// TIA Portal V19 export
DATA_BLOCK "BTrk"   // DB27
// stored: Access Published, MemoryReserve 100
   VAR RETAIN
      Last_B_ID : DInt;   // Ultimo ID asseggnato a una pezzo (Beam/Trave/Corrente)
   END_VAR
   VAR
      Empty : "BTrk_item";
   END_VAR
   VAR RETAIN
      EmptyLayer { S7_SetPoint := 'True'} : Array[1.."BTRK_LAYER_ITEMS"] of "BTrk_item";
      EmptyLayers : Array[1.."BTRK_LAYER_ITEMS"] of Struct
         Layer : Array[1.."BTRK_LAYER_ITEMS"] of "BTrk_item";
      END_STRUCT;
      A0301 : Struct
         Empty : Bool;
         MultipleOrders : Bool;
         O_ID : DInt;
         Beam_Qty : Int;
         Beam_Len : Real;
         Beam_W_A : Real;   // Dim. base (W) = Altezza in impilamento (A)
         Beam_H_B : Real;   // Dim. altezza (H) = base in impilamento (B)
         "B" : Array[1.."BTRK_A0301_ITEMS"] of "BTrk_item";   // Tracciamento travi su stazione primaria di assembleggio (capovolgimento semi-gusci)
      END_STRUCT;
      A0302_ENTRY : Struct
         Empty : Bool;
         MultipleOrders : Bool;
         O_ID : DInt;
         Beam_Qty : Int;
         Beam_Len : Real;
         Beam_W_A : Real;   // Dim. base (W) = Altezza in impilamento (A)
         Beam_H_B : Real;   // Dim. altezza (H) = base in impilamento (B)
         "B" : Array[1.."BTRK_A0302_ENTRY_ITEMS"] of "BTrk_item";   // Tracciamento travi su stazione finale di assemblaggio (chiusura bordi e allineamento longitudinale)
      END_STRUCT;
      A0302_EXIT : Struct
         Empty : Bool;
         MultipleOrders : Bool;
         O_ID : DInt;
         Beam_Qty : Int;
         Beam_Len : Real;
         Beam_W_A : Real;   // Dim. base (W) = Altezza in impilamento (A)
         Beam_H_B : Real;   // Dim. altezza (H) = base in impilamento (B)
         "B" : Array[1.."BTRK_A0302_EXIT_ITEMS"] of "BTrk_item";   // Tracciamento travi su stazione finale di assemblaggio (chiusura bordi e allineamento longitudinale)
      END_STRUCT;
      A03_EXIT_TOCHECK : Struct
         Empty : Bool;
         Beam_Qty : Int;
         "B" : Array[1.."BTRK_A03_EXIT_TOCHECK_ITEMS"] of "BTrk_item";   // Tracciamento travi su accumulo non conformi
      END_STRUCT;
      A0303 : Struct   // Tracciamento travi su stazione di preparazione pacco
         Preparation : Struct
            Empty : Bool;
            Completato : Bool;
            MultipleOrders : Bool;
            O_ID : DInt;
            BeamsPerLayer_Target : Int;   // Quanti pezzi per fare un layer
            Layers_Target : Int;   // Quanti layer
            Beam_Qty : Int;   // Da incrementare
            Beam_Len : Real;
            Beam_W_A : Real;   // Dim. base (W) = Altezza in impilamento (A)
            Beam_H_B : Real;   // Dim. altezza (H) = base in impilamento (B)
            "B" : "BTrk_item";
            Layer : Array[1.."BTRK_LAYER_ITEMS"] of "BTrk_item";
         END_STRUCT;
         Transfert : Struct
            Empty : Bool;
            MultipleOrders : Bool;
            O_ID : DInt;
            BeamsPerLayer_Target : Int;
            Layers_Target : Int;
            Beams_Qty : Int;
            Beams_Len : Real;
            Beams_W_A : Real;   // Dim. base (W) = Altezza in impilamento (A)
            Beams_H_B : Real;   // Dim. altezza (H) = base in impilamento (B)
            Layer { S7_SetPoint := 'True'} : Array[1.."BTRK_LAYER_ITEMS"] of "BTrk_item";
         END_STRUCT;
         Stacker : Struct
            Empty : Bool;
            Completato : Bool;
            MultipleOrders : Bool;
            O_ID : DInt;
            BeamsPerLayer_Target : Int;
            Layers_Target : Int;
            Layers_Qty : Int;
            Beams_Qty : Int;
            Beams_Len : Real;
            Beams_W_A : Real;   // Dim. base (W) = Altezza in impilamento (A)
            Beams_H_B : Real;   // Dim. altezza (H) = base in impilamento (B)
            Layers : Array[1.."BTRK_LAYER_ITEMS"] of Struct
               Layer : Array[1.."BTRK_LAYER_ITEMS"] of "BTrk_item";
            END_STRUCT;
         END_STRUCT;
      END_STRUCT;
      A0304 : Struct   // Tracciamento travi su stazione di scarico pacco
         Empty : Bool;
         MultipleOrders : Bool;
         NavettaInReggiatura : Bool;
         ReggiaturaConclusa : Bool;
         PaccoRimosso : Bool;
         AbilitazioneCancellazioneDatiPacco : Bool;
         O_ID : DInt;
         BeamsPerLayer_Target : Int;
         Layers_Target : Int;
         Layers_Qty : Int;
         Beams_Qty : Int;
         Beams_Len : Real;
         Beams_W_A : Real;   // Dim. base (W) = Altezza in impilamento (A)
         Beams_H_B : Real;   // Dim. altezza (H) = base in impilamento (B)
         Layers : Array[1.."BTRK_LAYER_ITEMS"] of Struct
            Layer : Array[1.."BTRK_LAYER_ITEMS"] of "BTrk_item";
         END_STRUCT;
      END_STRUCT;
   END_VAR
BEGIN
   // A0301."B"[1] : BTRK_A03_S1_Pos2_Lifter_Up
   // A0301."B"[2] : BTRK_A03_S1_Pos2_Lifter_Dwn
   // A0301."B"[3] : BTRK_A03_S1_Pos2_to_Pos3
   // A0301."B"[4] : BTRK_A03_S1_Pos3_Entry
   // A0301."B"[5] : BTRK_A03_S1_Pos3_Exit
   // A0301."B"[6] : BTRK_A03_S1_Pos3_to_Pos4
   // A0301."B"[7] : BTRK_A03_S1_Pos4_Entry
   // A0301."B"[8] : BTRK_A03_S1_Pos4_Exit
   // A0301."B"[9] : BTRK_A03_S1_Pos4_to_LateralAligner
   // A0301."B"[10] : BTRK_A03_S1_LateralAligner_Home_Pos
   // A0301."B"[11] : BTRK_A03_S1_LateralAligner_Work_Pos
   // A0301."B"[12] : BTRK_A03_S1_Free12
   // A0301."B"[13] : BTRK_A03_S1_Free13
   // A0301."B"[14] : BTRK_A03_S1_Free14
   // A0301."B"[15] : BTRK_A03_S1_Free15
   // A0301."B"[16] : BTRK_A03_S1_Free16
   // A0301."B"[17] : BTRK_A03_S1_Free17
   // A0301."B"[18] : BTRK_A03_S1_Free18
   // A0301."B"[19] : BTRK_A03_S1_Free19
   // A0301."B"[20] : BTRK_A03_S1_Free20
   // A0302_ENTRY."B"[1] : BTRK_A03_S2_Pusher_Home_Lift_dwn
   // A0302_ENTRY."B"[2] : BTRK_A03_S2_Pusher_Home_Lift_Up
   // A0302_ENTRY."B"[3] : BTRK_A03_S2_Pusher_Working_Range
   // A0302_ENTRY."B"[4] : BTRK_A03_S2_Joining_Entry
   // A0302_ENTRY."B"[5] : BTRK_A03_S2_Joining_Exit
   // A0302_ENTRY."B"[6] : BTRK_A03_S2_Roller
   // A0302_ENTRY."B"[7] : BTRK_A03_S2_Roller_to_Centering
   // A0302_EXIT."B"[1] : BTRK_A03_S2_Pusher_Home_Lift_dwn
   // A0302_EXIT."B"[2] : BTRK_A03_S2_Pusher_Home_Lift_Up
   // A0302_EXIT."B"[3] : BTRK_A03_S2_Pusher_Working_Range
   // A0302_EXIT."B"[4] : BTRK_A03_S2_Joining_Entry
   // A0302_EXIT."B"[5] : BTRK_A03_S2_Joining_Exit
   // A0302_EXIT."B"[6] : BTRK_A03_S2_Roller
   // A0302_EXIT."B"[7] : BTRK_A03_S2_Roller_to_Centering
   // A0302_EXIT."B"[8] : BTRK_A03_S2_Centering
   // A0302_EXIT."B"[9] : BTRK_A03_S2_Centering_to_Deviator
   // A0302_EXIT."B"[10] : BTRK_A03_S2_Deviator_To_EXIT
END_DATA_BLOCK
